Universal Robots PolyScope program: LAB4.urp

Program LAB4 (installation=default directory=/home/ur/ursim-current/programs createdIn=3.12.1.90940 lastSavedIn=3.12.1.90940 robotSerialNumber=2018339999)
Calibrated DH parameters: a=[0, -0.24365, -0.21325, 0, 0, 0]; d=[0.1519, 0, 0, 0.11235, 0.08535, 0.0819]; alpha=[1.570796, 0, 0, 1.570796, -1.570796, 0]; deltaTheta=[0, 0, 0, 0, 0, 0]
BeforeStart
  startpos := p[0.1, -0.3, 0.17, -3.14, 0, 0]
  pickup := p[0.3, -0.21, 0.12, -3.14, 0, 0]
  delivery := p[-0.1, -0.35, 0.024, -3.14, 0, 0]
  delivery_h := pose_add(delivery, p[0,0,0.146,0,0,0])
  pickup_h := pose_add(pickup, p[0,0,0.05,0,0,0])
Robot Program (runOnlyOnce=true)
  Script file /home/ur/ursim-current/programs/move.script
    | movel(startpos)
    | 
    | i = 0
    | z_ret = 0.024
    | 
    | while i < 5:
    | 	movel(pickup_h)
    | 	movel(pickup)
    | 
    | 	set_digital_out(0, True)
    | 	sleep(0.5)
    | 
    | 	movel(pickup_h)
    | 	movel(delivery_h)
    | 	movel(delivery)
    | 
    | 	set_digital_out(0, False)
    | 	sleep(0.5)
    | 
    | 	movel(delivery_h)
    | 
    | 	i = i+1
    | 	pickup = pose_add(pickup,p[0,0,-z_ret,0,0,0])
    | 	delivery = pose_add(delivery,p[0,0,z_ret,0,0,0])
    | end
    | 
    | movel(startpos)
